# EPICS autosave request: ipApp/Db/ADAM_4018p_chan_settings.req
$(P)$(R):tc$(C).DESC
$(P)$(R):tc$(C).SCAN
$(P)$(R):temp$(C).DESC
$(P)$(R):unit$(C).VAL
